FUNCTION_BLOCK IntegrationTestSuite
VAR
	StubAxis : AXIS_REF;
	gearSlave : AXIS_REF;
	TestAxis : Axis_Base(StubAxis);
	gearTestAxis : Axis_Base(gearSlave);
	iAxisBase : I_AxisBase := TestAxis;
	iJog : I_Jog := TestAxis;
	iAxisStatus : I_Status := TestAxis;
	iPosition : I_Position := TestAxis;
	iVelo : I_Velocity := TestAxis;
	gearOperation : GearAxes := (Master := TestAxis, Slave := gearTestAxis);
	Enable: BOOL;
	MOVETO: BOOL;
	MOVETWO: BOOL;
	MOVEREL : BOOL;
	DISABLE: BOOL;
	SETBUFFER: BOOL;
	CONVEYOR: BOOL;
	JOGSLOW: BOOL;
	JOGFAST: BOOL;
	HALT: BOOL;
	MODULO : BOOL;
	VelocityDemand : LREAL := 100.0;
	Pos_Dist : LREAL := 10.0;
	Mod_Pos : LREAL := 230.0;
	GEAR: BOOL;
	checkflag : BOOL;
	istartCounter: INT;
	ioperatCounter : INT;
	stationaryTest1: BOOL;
	stationaryTest2: BOOL;
END_VAR

IF Enable THEN
	IF succeeded(iAxisBase.EnableAxis(FALSE, FALSE)) AND SUCCEEDED(gearTestAxis.EnableAxis(FALSE,FALSE)) THEN
		Enable := FALSE;
	END_IF
END_IF
 IF checkflag THEN
	 istartCounter := istartCounter + 1;
 END_IF

IF iAxisBase.Operating THEN
	checkflag := FALSE;
	ioperatCounter := ioperatCounter + 1;
END_IF

IF MOVETO THEN
	IF SUCCEEDED(iPosition.MoveToPosition(1000.0,100.0)) THEN
		checkflag := TRUE;
		MOVETO := FALSE;
	END_IF
END_IF

IF SETBUFFER THEN
	SETBUFFER := FALSE;
	TestAxis.BufferMode := MC_BufferMode.MC_BlendingLow;
	
END_IF

IF MOVETWO THEN
	IF SUCCEEDED(iPosition.MoveToPosition(1200.0,VelocityDemand)) THEN
		MOVETWO := FALSE;
	END_IF
END_IF

IF MOVEREL THEN
	IF succeeded(iPosition.MoveByDistance(Pos_Dist,VelocityDemand)) THEN
		MOVEREL := FALSE;
	END_IF
END_IF

IF MODULO THEN
	IF SUCCEEDED(iPosition.MoveToModuloPosition(Mod_Pos,VelocityDemand)) THEN
		MODULO := FALSE;
	END_IF
END_IF

IF HALT THEN
	IF SUCCEEDED(iAxisBase.HaltAxis()) THEN
		HALT := FALSE;
	END_IF
END_IF

IF DISABLE THEN
	IF SUCCEEDED(iAxisBase.DisableAxis()) AND SUCCEEDED(gearTestAxis.DisableAxis()) THEN
		DISABLE := FALSE;
	END_IF
END_IF

IF GEAR THEN
	IF SUCCEEDED(gearOperation.GearIn()) THEN
		GEAR := FALSE;
	END_IF
END_IF

IF CONVEYOR THEN
	IF SUCCEEDED(iVelo.MoveAtVelocity(MC_Direction.MC_Positive_Direction, VelocityDemand)) THEN
		CONVEYOR := FALSE;
	END_IF
END_IF

IF JOGSLOW THEN
	iJog.JogSlow(FALSE);
END_IF

IF JOGFAST THEN
	iJog.JogFast(TRUE);
END_IF

stationaryTest1 := TestAxis.IsStationary;
stationaryTest2 := gearTestAxis.IsStationary;

TestAxis.Cycle();
gearTestAxis.Cycle();
gearOperation.Cycle();

END_FUNCTION_BLOCK

(* stored: Version 1.1.0.1
   POU IntegrationTestSuite: Id {69bc61fe-8999-4914-8ef6-bb0c95ff7655}, SpecialFunc None *)
